(* CoDeSys 2.3.9.55 project: PLC rolety modbus.pro *)
(* Libraries: Targets\WAGO\Libraries\32_Bit\SysLibRtc.lib 8.11.10 12:37:48, Targets\WAGO\Libraries\32_Bit\Visu_Scheduler_03_e.lib 27.1.21 14:42:06, SysLibFile.lib 8.11.10 12:37:48, mod_com.lib 8.11.10 12:37:48, Targets\WAGO\Libraries\32_Bit\Scheduler_03.lib 27.1.21 14:42:05, Targets\WAGO\Libraries\32_Bit\oscat_building_100.lib 24.3.25 16:40:53, Building_common.lib 28.9.15 13:45:22, Targets\WAGO\Libraries\32_Bit\oscat_basic_333.lib 24.3.25 16:48:54, Standard.lib 8.11.10 12:37:48, SYSLIBCALLBACK.LIB 8.11.10 12:37:48 *)

(* PLC configuration (modules and I/O channels)
IN1 AT %IX0.0 [BOOLOnX_I] Biuro
IN2 AT %IX0.1 [BOOLOnX_I] Garaz
IN3 AT %IX0.2 [BOOLOnX_I] Jadalnia
IN4 AT %IX0.3 [BOOLOnX_I] Kuchnia duze
IN5 AT %IX0.4 [BOOLOnX_I] Kuchnia male
IN6 AT %IX0.5 [BOOLOnX_I] Lazienka duza
IN7 AT %IX0.6 [BOOLOnX_I] Salon duze 1
IN8 AT %IX0.7 [BOOLOnX_I] Salon duze 2
IN9 AT %IX0.8 [BOOLOnX_I] Salon taras
IN10 AT %IX0.9 [BOOLOnX_I] Schody
IN11 AT %IX0.10 [BOOLOnX_I] Sypialnia
IN12 AT %IX0.11 [BOOLOnX_I] Taras drzwi
IN13 AT %IX0.12 [BOOLOnX_I] Warsztat
IN14 AT %IX0.13 [BOOLOnX_I] rezerwa
IN15 AT %IX0.14 [BOOLOnX_I] Otworz wszystkie
IN16 AT %IX0.15 [BOOLOnX_I] Zamknij wszystkie
0750-0513 2 DO 250V AC 2.0A Rel 2NO (PotFree) [Type_10_2_Channels] node 2, in %IB1 out %QB0 {INTTypePAAssignment = PLC; INTTypeModule = plugged}
  OUTO1 AT %QX0.0 [BOOLOnX_Q] Biuro otwórz
  OUTC1 AT %QX0.1 [BOOLOnX_Q] Biuro zamknij
0750-0513 2 DO 250V AC 2.0A Rel 2NO (PotFree) [Type_10_2_Channels] node 3, in %IB2 out %QB0 {INTTypePAAssignment = PLC; INTTypeModule = plugged}
  OUTO2 AT %QX0.2 [BOOLOnX_Q] Garaz otwórz
  OUTC2 AT %QX0.3 [BOOLOnX_Q] Garaz zamknij
0750-0513 2 DO 250V AC 2.0A Rel 2NO (PotFree) [Type_10_2_Channels] node 4, in %IB2 out %QX0.2 {INTTypePAAssignment = PLC; INTTypeModule = plugged}
  OUTO3 AT %QX0.4 [BOOLOnX_Q] Jadalnia otwórz
  OUTC3 AT %QX0.5 [BOOLOnX_Q] Jadalnia zamknij
0750-0513 2 DO 250V AC 2.0A Rel 2NO (PotFree) [Type_10_2_Channels] node 5, in %IB2 out %QX0.4 {INTTypePAAssignment = PLC; INTTypeModule = plugged}
  OUTO4 AT %QX0.6 [BOOLOnX_Q] Kuchnia duze otwórz
  OUTC4 AT %QX0.7 [BOOLOnX_Q] Kuchnia duze zamknij
0750-0513 2 DO 250V AC 2.0A Rel 2NO (PotFree) [Type_10_2_Channels] node 6, in %IB2 out %QX0.6 {INTTypePAAssignment = PLC; INTTypeModule = plugged}
  OUTO5 AT %QX0.8 [BOOLOnX_Q] Kuchnia male otwórz
  OUTC5 AT %QX0.9 [BOOLOnX_Q] Kuchnia male zamknij
0750-0513 2 DO 250V AC 2.0A Rel 2NO (PotFree) [Type_10_2_Channels] node 7, in %IB2 out %QB1 {INTTypePAAssignment = PLC; INTTypeModule = plugged}
  OUTO6 AT %QX0.10 [BOOLOnX_Q] Lazienka duza otwórz
  OUTC6 AT %QX0.11 [BOOLOnX_Q] Lazienka duza zamknij
0750-0513 2 DO 250V AC 2.0A Rel 2NO (PotFree) [Type_10_2_Channels] node 8, in %IB2 out %QX0.10 {INTTypePAAssignment = PLC; INTTypeModule = plugged}
  OUTO7 AT %QX0.12 [BOOLOnX_Q] Salon duze 1 otwórz
  OUTC7 AT %QX0.13 [BOOLOnX_Q] Salon duze 1 zamknij
0750-0513 2 DO 250V AC 2.0A Rel 2NO (PotFree) [Type_10_2_Channels] node 9, in %IB2 out %QX0.12 {INTTypePAAssignment = PLC; INTTypeModule = plugged}
  OUTO8 AT %QX0.14 [BOOLOnX_Q] Salon duze 2 otwórz
  OUTC8 AT %QX0.15 [BOOLOnX_Q] Salon duze 2 zamknij
0750-0513 2 DO 250V AC 2.0A Rel 2NO (PotFree) [Type_10_2_Channels] node 10, in %IB2 out %QX0.14 {INTTypePAAssignment = PLC; INTTypeModule = plugged}
  OUTO9 AT %QX1.0 [BOOLOnX_Q] Salon taras otwórz
  OUTC9 AT %QX1.1 [BOOLOnX_Q] Salon taras zamknij
0750-0513 2 DO 250V AC 2.0A Rel 2NO (PotFree) [Type_10_2_Channels] node 11, in %IB2 out %QB2 {INTTypePAAssignment = PLC; INTTypeModule = plugged}
  OUTO10 AT %QX1.2 [BOOLOnX_Q] Schody otwórz
  OUTC10 AT %QX1.3 [BOOLOnX_Q] Schody zamknij
0750-0513 2 DO 250V AC 2.0A Rel 2NO (PotFree) [Type_10_2_Channels] node 12, in %IB2 out %QX1.2 {INTTypePAAssignment = PLC; INTTypeModule = plugged}
  OUTO11 AT %QX1.4 [BOOLOnX_Q] Sypialnia otwórz
  OUTC11 AT %QX1.5 [BOOLOnX_Q] Sypialnia zamknij
0750-0513 2 DO 250V AC 2.0A Rel 2NO (PotFree) [Type_10_2_Channels] node 13, in %IB2 out %QX1.4 {INTTypePAAssignment = PLC; INTTypeModule = plugged}
  OUTO12 AT %QX1.6 [BOOLOnX_Q] Taras otwórz
  OUTC12 AT %QX1.7 [BOOLOnX_Q] Taras zamknij
0750-0513 2 DO 250V AC 2.0A Rel 2NO (PotFree) [Type_10_2_Channels] node 14, in %IB2 out %QX1.6 {INTTypePAAssignment = PLC; INTTypeModule = plugged}
  OUTO13 AT %QX1.8 [BOOLOnX_Q] Warsztat otwórz
  OUTC13 AT %QX1.9 [BOOLOnX_Q] Warsztat zamknij
Fieldbus variables [FB_VARS] node 1, in %IB0 out %QB0
Flag variables [FLAG_VARS] node 2, in %IB0 out %QB0
Modbus-Master [MB_MASTER] node 3, in %IB0 out %QB0
*)

(* Task configuration *)
TASK Main (PRIORITY := 1); (* freewheeling *)
	PLC_PRG();
END_TASK
TASK ReadClock (PRIORITY := 10, INTERVAL := T#1000ms);
	ReadClock();
END_TASK

(* Global variable list: Global_Variables *)
VAR_GLOBAL
  CURRENT_TIME : DATE_AND_TIME;
END_VAR

(* POU PLC_PRG, ST *)
PROGRAM PLC_PRG
VAR
	(*programator tygodniowy *)
	Enable_Schedulers : BOOL := TRUE;
	Scheduler_Blind_1, Scheduler_Blind_2 : FbScheduleWeekly;
  	Scheduler_Blind_1_ON, Scheduler_Blind_2_ON : R_TRIG;
  	Scheduler_Blind_1_OFF, Scheduler_Blind_2_OFF : F_TRIG;
 	Blinds_UP, Blinds_DN : BOOL;
	(* Przyciski long/short do sterowania roletami  - 1 sec. *)
	LongShort_IN1, LongShort_IN2, LongShort_IN3, LongShort_IN4, LongShort_IN5, LongShort_IN6, LongShort_IN7, LongShort_IN8, LongShort_IN9,  LongShort_IN10,  LongShort_IN11,  LongShort_IN12,  LongShort_IN13, LongShort_IN15, LongShort_IN16 : Fb_ShortLong := (uiT_10tel_s := 10, uiTL_10tel_s := 1, uiTS_10tel_s := 1);
	(*Przyciski podwojny klik*)
	Double_IN1, Double_IN2, Double_IN3, Double_IN4, Double_IN5, Double_IN6, Double_IN7, Double_IN8, Double_IN9,  Double_IN10,  Double_IN11,  Double_IN12,  Double_IN13 : Fb_Click;
	(* Wizualizacje - Rolety *)
	VIS_Blind_1_UP,  VIS_Blind_1_DN, VIS_1_wlacz, VIS_Blind_1_SHADE : BOOL;
	VIS_Blind_2_UP,  VIS_Blind_2_DN, VIS_2_wlacz, VIS_Blind_2_SHADE : BOOL;
	VIS_Blind_3_UP,  VIS_Blind_3_DN, VIS_3_wlacz, VIS_Blind_3_SHADE : BOOL;
	VIS_Blind_4_UP,  VIS_Blind_4_DN, VIS_4_wlacz, VIS_Blind_4_SHADE : BOOL;
	VIS_Blind_5_UP,  VIS_Blind_5_DN, VIS_5_wlacz, VIS_Blind_5_SHADE : BOOL;
	VIS_Blind_6_UP,  VIS_Blind_6_DN, VIS_6_wlacz, VIS_Blind_6_SHADE : BOOL;
	VIS_Blind_7_UP,  VIS_Blind_7_DN, VIS_7_wlacz, VIS_Blind_7_SHADE : BOOL;
	VIS_Blind_8_UP,  VIS_Blind_8_DN, VIS_8_wlacz, VIS_Blind_8_SHADE : BOOL;
	VIS_Blind_9_UP,  VIS_Blind_9_DN, VIS_9_wlacz, VIS_Blind_9_SHADE : BOOL;
	VIS_Blind_10_UP,  VIS_Blind_10_DN, VIS_10_wlacz, VIS_Blind_10_SHADE : BOOL;
	VIS_Blind_11_UP,  VIS_Blind_11_DN, VIS_11_wlacz, VIS_Blind_11_SHADE : BOOL;
	VIS_Blind_12_UP,  VIS_Blind_12_DN, VIS_12_wlacz, VIS_Blind_12_SHADE : BOOL;
	VIS_Blind_13_UP,  VIS_Blind_13_DN, VIS_13_wlacz, VIS_Blind_13_SHADE : BOOL;
	(* przyciski otwórz/zamknij wszystkie *)
 	VIS_ALL_UP,  VIS_ALL_DN  : BOOL; (* do sterowania z wizualizacji *)
	(*deklaracje modbus*)
	VIS_OUT1 AT %MX294.0: BOOL;
	VIS_OUT2 AT %MX295.0: BOOL;
	VIS_OUT3 AT %MX296.0: BOOL;
	VIS_OUT4 AT %MX297.0: BOOL;
	VIS_OUT5 AT %MX298.0: BOOL;
	VIS_OUT6 AT %MX299.0: BOOL;
	VIS_OUT7 AT %MX300.0: BOOL;
	VIS_OUT8 AT %MX301.0: BOOL;
	VIS_OUT9 AT %MX302.0: BOOL;
	VIS_OUT10 AT %MX303.0: BOOL;
	VIS_OUT11 AT %MX304.0: BOOL;
	VIS_OUT12 AT %MX305.0: BOOL;
	VIS_OUT13 AT %MX306.0: BOOL;
	VIS_OUT14 AT %MX307.0: BOOL;
	VIS_OUT15 AT %MX308.0: BOOL;
	VIS_OUT16 AT %MX309.0: BOOL;
	VIS_OUT17 AT %MX310.0: BOOL;
	VIS_OUT18 AT %MX311.0: BOOL;
	VIS_OUT19 AT %MX312.0: BOOL;
	VIS_OUT20 AT %MX313.0: BOOL;
	VIS_OUT21 AT %MX314.0: BOOL;
	VIS_OUT22 AT %MX315.0: BOOL;
	VIS_OUT23 AT %MX316.0: BOOL;
	VIS_OUT24 AT %MX317.0: BOOL;
	VIS_OUT25 AT %MX318.0: BOOL;
	VIS_OUT26 AT %MX319.0: BOOL;
	VIS_OUT_ALL_UP AT %MX326.0: BOOL;
	VIS_OUT_ALL_DN AT %MX327.0: BOOL;
END_VAR
VAR RETAIN PERSISTENT
	(* Programator tygodniowy *)
	Data_Blind_1, Data_Blind_2 : typScheduleWeekly;
	(* Rolety *)
	Input_Blind_1: BLIND_INPUT := (PI := 150, MAX_RUNTIME := T#20s, MANUAL_TIMEOUT := t#60m, MASTER_MODE := TRUE);
	Control_Blind_1 : BLIND_CONTROL_S := (T_UP := T#17s, T_DN := T#17s);
	Input_Blind_2: BLIND_INPUT := (PI := 150, MAX_RUNTIME := T#35s, MANUAL_TIMEOUT := t#60m, MASTER_MODE := TRUE);
	Control_Blind_2 : BLIND_CONTROL_S := (T_UP := T#30s, T_DN := T#30s);
	Input_Blind_3: BLIND_INPUT := (PI := 150, MAX_RUNTIME := T#35s, MANUAL_TIMEOUT := t#60m, MASTER_MODE := TRUE);
	Control_Blind_3 : BLIND_CONTROL_S := (T_UP := T#30s, T_DN := T#30s);
	Input_Blind_4: BLIND_INPUT := (PI := 150, MAX_RUNTIME := T#20s, MANUAL_TIMEOUT := t#60m, MASTER_MODE := TRUE);
	Control_Blind_4 : BLIND_CONTROL_S := (T_UP := T#17s, T_DN := T#17s);
	Input_Blind_5: BLIND_INPUT := (PI := 150, MAX_RUNTIME := T#20s, MANUAL_TIMEOUT := t#60m, MASTER_MODE := TRUE);
	Control_Blind_5 : BLIND_CONTROL_S := (T_UP := T#17s, T_DN := T#17s);
	Input_Blind_6: BLIND_INPUT := (PI := 150, MAX_RUNTIME := T#35s, MANUAL_TIMEOUT := t#60m, MASTER_MODE := TRUE);
	Control_Blind_6 : BLIND_CONTROL_S := (T_UP := T#30s, T_DN := T#30s);
	Input_Blind_7: BLIND_INPUT := (PI := 150, MAX_RUNTIME := T#35s, MANUAL_TIMEOUT := t#60m, MASTER_MODE := TRUE);
	Control_Blind_7 : BLIND_CONTROL_S := (T_UP := T#30s, T_DN := T#30s);
	Input_Blind_8: BLIND_INPUT := (PI := 150, MAX_RUNTIME := T#35s, MANUAL_TIMEOUT := t#60m, MASTER_MODE := TRUE);
	Control_Blind_8 : BLIND_CONTROL_S := (T_UP := T#30s, T_DN := T#30s);
	Input_Blind_9: BLIND_INPUT := (PI := 150, MAX_RUNTIME := T#35s, MANUAL_TIMEOUT := t#60m, MASTER_MODE := TRUE);
	Control_Blind_9 : BLIND_CONTROL_S := (T_UP := T#30s, T_DN := T#30s);
	Input_Blind_10: BLIND_INPUT := (PI := 150, MAX_RUNTIME := T#20s, MANUAL_TIMEOUT := t#60m, MASTER_MODE := TRUE);
	Control_Blind_10 : BLIND_CONTROL_S := (T_UP := T#17s, T_DN := T#17s);
	Input_Blind_11: BLIND_INPUT := (PI := 150, MAX_RUNTIME := T#20s, MANUAL_TIMEOUT := t#60m, MASTER_MODE := TRUE);
	Control_Blind_11 : BLIND_CONTROL_S := (T_UP := T#17s, T_DN := T#17s);
	Input_Blind_12: BLIND_INPUT := (PI := 150, MAX_RUNTIME := T#35s, MANUAL_TIMEOUT := t#60m, MASTER_MODE := TRUE);
	Control_Blind_12 : BLIND_CONTROL_S := (T_UP := T#30s, T_DN := T#30s);
	Input_Blind_13: BLIND_INPUT := (PI := 150, MAX_RUNTIME := T#35s, MANUAL_TIMEOUT := t#60m, MASTER_MODE := TRUE);
	Control_Blind_13 : BLIND_CONTROL_S := (T_UP := T#30s, T_DN := T#30s);
	Input_Blind_ALL: BLIND_INPUT := (PI := 150, MAX_RUNTIME := T#35s, MANUAL_TIMEOUT := t#60m, MASTER_MODE := TRUE);
	Control_Blind_ALL : BLIND_CONTROL_S := (T_UP := T#30s, T_DN := T#30s);
END_VAR
(*bloki zarzadzajace timerami*)
Scheduler_Blind_1(xEnable := Enable_Schedulers, dtActualTime := CURRENT_TIME, typScheduleWeekly := Data_Blind_1);
Scheduler_Blind_2(xEnable := Enable_Schedulers, dtActualTime := CURRENT_TIME, typScheduleWeekly := Data_Blind_2);
(*wykrywanie wlaczenia/wylaczenia bloków timerów*)
Scheduler_Blind_1_ON(CLK := Scheduler_Blind_1.xSwitchChannel);
Scheduler_Blind_1_OFF(CLK := Scheduler_Blind_1.xSwitchChannel);
Scheduler_Blind_2_ON(CLK := Scheduler_Blind_2.xSwitchChannel);
Scheduler_Blind_2_OFF(CLK := Scheduler_Blind_2.xSwitchChannel);
(*sumowanie impulsów ON/OFF/Otworz-zamknij-wszystkie*)
Blinds_UP := Scheduler_Blind_1_ON.Q OR Scheduler_Blind_2_ON.Q OR VIS_ALL_UP;
Blinds_DN := Scheduler_Blind_1_OFF.Q OR Scheduler_Blind_2_OFF.Q OR VIS_ALL_DN;
(* ---------- przepianie rejestrow wejsciowych i wyjsciowych do podgladu --------------- *)
%MW100 := %IW0;
%MW200 := %QW0;
(* ---------- przyciski KRÓTKI / DLUGI --------------- *)
LongShort_IN1( xSwitch := IN1 );
LongShort_IN2( xSwitch := IN2 );
LongShort_IN3( xSwitch := IN3 );
LongShort_IN4( xSwitch := IN4 );
LongShort_IN5( xSwitch := IN5 );
LongShort_IN6( xSwitch := IN6 );
LongShort_IN7( xSwitch := IN7 );
LongShort_IN8( xSwitch := IN8 );
LongShort_IN9( xSwitch := IN9 );
LongShort_IN10( xSwitch := IN10 );
LongShort_IN11( xSwitch := IN11 );
LongShort_IN12( xSwitch := IN12 );
LongShort_IN13( xSwitch := IN13 );
LongShort_IN15( xSwitch := IN15 );
LongShort_IN16( xSwitch := IN16 );
(*Przyciski double*)
Double_IN1( xSwitch := IN1 );
Double_IN2( xSwitch := IN2 );
Double_IN3( xSwitch := IN3 );
Double_IN4( xSwitch := IN4 );
Double_IN5( xSwitch := IN5 );
Double_IN6( xSwitch := IN6 );
Double_IN7( xSwitch := IN7 );
Double_IN8( xSwitch := IN8 );
Double_IN9( xSwitch := IN9 );
Double_IN10( xSwitch := IN10 );
Double_IN11( xSwitch := IN11 );
Double_IN12( xSwitch := IN12 );
Double_IN13( xSwitch := IN13 );
(* ------------- ROLETY ------------------*)
(*Roleta Biuro*)
Input_Blind_1(
S1 := LongShort_IN1.xShort OR LongShort_IN15.xLong OR VIS_Blind_1_UP OR Blinds_UP AND VIS_1_wlacz OR VIS_OUT_ALL_UP AND VIS_1_wlacz OR VIS_OUT1,
S2 := LongShort_IN1.xLong OR LongShort_IN16.xLong OR VIS_Blind_1_DN OR Blinds_DN AND VIS_1_wlacz OR VIS_OUT_ALL_DN AND VIS_1_wlacz OR VIS_OUT2,
IN := VIS_Blind_1_SHADE OR Double_IN1.xDouble, POS := Control_Blind_1.POS
);
Control_Blind_1(
UP := Input_Blind_1.QU,
DN := Input_Blind_1.QD,
S_IN := Input_Blind_1.STATUS,
pi := Input_Blind_1.PO
);
OUTO1 := Control_Blind_1.MU;
OUTC1 := Control_Blind_1.MD;
(*Roleta Garaz*)
Input_Blind_2(
S1 := LongShort_IN2.xShort OR LongShort_IN15.xLong OR VIS_Blind_2_UP OR Blinds_UP AND VIS_2_wlacz OR VIS_OUT_ALL_UP AND VIS_2_wlacz OR VIS_OUT3,
S2 := LongShort_IN2.xLong OR LongShort_IN16.xLong OR VIS_Blind_2_DN OR Blinds_DN AND VIS_2_wlacz OR VIS_OUT_ALL_DN AND VIS_2_wlacz OR VIS_OUT4,
IN := VIS_Blind_2_SHADE OR Double_IN2.xDouble, POS := Control_Blind_2.POS
);
Control_Blind_2(
UP := Input_Blind_2.QU,
DN := Input_Blind_2.QD,
S_IN := Input_Blind_2.STATUS,
pi := Input_Blind_2.PO
);
OUTO2 := Control_Blind_2.MU;
OUTC2 := Control_Blind_2.MD;
(*Roleta Jadalnia*)
Input_Blind_3(
S1 := LongShort_IN3.xShort OR LongShort_IN15.xLong OR VIS_Blind_3_UP OR Blinds_UP AND VIS_3_wlacz OR VIS_OUT_ALL_UP AND VIS_3_wlacz OR VIS_OUT5,
S2 := LongShort_IN3.xLong OR LongShort_IN16.xLong OR VIS_Blind_3_DN OR Blinds_DN AND VIS_3_wlacz OR VIS_OUT_ALL_DN AND VIS_3_wlacz OR VIS_OUT6,
IN := VIS_Blind_3_SHADE OR Double_IN3.xDouble, POS := Control_Blind_3.POS
);
Control_Blind_3(
UP := Input_Blind_3.QU,
DN := Input_Blind_3.QD,
S_IN := Input_Blind_3.STATUS,
pi := Input_Blind_3.PO
);
OUTO3 := Control_Blind_3.MU;
OUTC3 := Control_Blind_3.MD;
(*Roleta Kuchnia duze*)
Input_Blind_4(
S1 := LongShort_IN4.xShort OR LongShort_IN15.xLong OR VIS_Blind_4_UP OR Blinds_UP AND VIS_4_wlacz OR VIS_OUT_ALL_UP AND VIS_4_wlacz OR VIS_OUT7,
S2 := LongShort_IN4.xLong OR LongShort_IN16.xLong OR VIS_Blind_4_DN OR Blinds_DN AND VIS_4_wlacz OR VIS_OUT_ALL_DN AND VIS_4_wlacz OR VIS_OUT8,
IN := VIS_Blind_4_SHADE OR Double_IN4.xDouble, POS := Control_Blind_4.POS
);
Control_Blind_4(
UP := Input_Blind_4.QU,
DN := Input_Blind_4.QD,
S_IN := Input_Blind_4.STATUS,
pi := Input_Blind_4.PO
);
OUTO4 := Control_Blind_4.MU;
OUTC4 := Control_Blind_4.MD;
(*Roleta Kuchnia male*)
Input_Blind_5(
S1 := LongShort_IN5.xShort OR LongShort_IN15.xLong OR VIS_Blind_5_UP OR Blinds_UP AND VIS_5_wlacz OR VIS_OUT_ALL_UP AND VIS_5_wlacz OR VIS_OUT9,
S2 := LongShort_IN5.xLong OR LongShort_IN16.xLong OR VIS_Blind_5_DN OR Blinds_DN AND VIS_5_wlacz OR VIS_OUT_ALL_DN AND VIS_5_wlacz OR VIS_OUT10,
IN := VIS_Blind_5_SHADE OR Double_IN5.xDouble, POS := Control_Blind_5.POS
);
Control_Blind_5(
UP := Input_Blind_5.QU,
DN := Input_Blind_5.QD,
S_IN := Input_Blind_5.STATUS,
pi := Input_Blind_5.PO
);
OUTO5 := Control_Blind_5.MU;
OUTC5 := Control_Blind_5.MD;
(*Roleta Lazienka duza*)
Input_Blind_6(
S1 := LongShort_IN6.xShort OR LongShort_IN15.xLong OR VIS_Blind_6_UP OR Blinds_UP AND VIS_6_wlacz OR VIS_OUT_ALL_UP AND VIS_6_wlacz OR VIS_OUT11,
S2 := LongShort_IN6.xLong OR LongShort_IN16.xLong OR VIS_Blind_6_DN OR Blinds_DN AND VIS_6_wlacz OR VIS_OUT_ALL_DN AND VIS_6_wlacz OR VIS_OUT12,
IN := VIS_Blind_6_SHADE OR Double_IN6.xDouble, POS := Control_Blind_6.POS
);
Control_Blind_6(
UP := Input_Blind_6.QU,
DN := Input_Blind_6.QD,
S_IN := Input_Blind_6.STATUS,
pi := Input_Blind_6.PO
);
OUTO6 := Control_Blind_6.MU;
OUTC6 := Control_Blind_6.MD;
(*Roleta Salon duze 1*)
Input_Blind_7(
S1 := LongShort_IN7.xShort OR LongShort_IN15.xLong OR VIS_Blind_7_UP OR Blinds_UP AND VIS_7_wlacz OR VIS_OUT_ALL_UP AND VIS_7_wlacz OR VIS_OUT13,
S2 := LongShort_IN7.xLong OR LongShort_IN16.xLong OR VIS_Blind_7_DN OR Blinds_DN AND VIS_7_wlacz OR VIS_OUT_ALL_DN AND VIS_7_wlacz OR VIS_OUT14,
IN := VIS_Blind_7_SHADE OR Double_IN7.xDouble, POS := Control_Blind_7.POS
);
Control_Blind_7(
UP := Input_Blind_7.QU,
DN := Input_Blind_7.QD,
S_IN := Input_Blind_7.STATUS,
pi := Input_Blind_7.PO
);
OUTO7 := Control_Blind_7.MU;
OUTC7 := Control_Blind_7.MD;
(*Roleta Salon duze 2*)
Input_Blind_8(
S1 := LongShort_IN8.xShort OR LongShort_IN15.xLong OR VIS_Blind_8_UP OR Blinds_UP AND VIS_8_wlacz OR VIS_OUT_ALL_UP AND VIS_8_wlacz OR VIS_OUT15,
S2 := LongShort_IN8.xLong OR LongShort_IN16.xLong OR VIS_Blind_8_DN OR Blinds_DN AND VIS_8_wlacz OR VIS_OUT_ALL_DN AND VIS_8_wlacz OR VIS_OUT16,
IN := VIS_Blind_8_SHADE OR Double_IN8.xDouble, POS := Control_Blind_8.POS
);
Control_Blind_8(
UP := Input_Blind_8.QU,
DN := Input_Blind_8.QD,
S_IN := Input_Blind_8.STATUS,
pi := Input_Blind_8.PO
);
OUTO8 := Control_Blind_8.MU;
OUTC8 := Control_Blind_8.MD;
(*Roleta  Salon taras*)
Input_Blind_9(
S1 := LongShort_IN9.xShort OR LongShort_IN15.xLong OR VIS_Blind_9_UP OR Blinds_UP AND VIS_9_wlacz OR VIS_OUT_ALL_UP AND VIS_9_wlacz OR VIS_OUT17,
S2 := LongShort_IN9.xLong OR LongShort_IN16.xLong OR VIS_Blind_9_DN OR Blinds_DN AND VIS_9_wlacz OR VIS_OUT_ALL_DN AND VIS_9_wlacz OR VIS_OUT18,
IN := VIS_Blind_9_SHADE OR Double_IN9.xDouble, POS := Control_Blind_9.POS
);
Control_Blind_9(
UP := Input_Blind_9.QU,
DN := Input_Blind_9.QD,
S_IN := Input_Blind_9.STATUS,
pi := Input_Blind_9.PO
);
OUTO9 := Control_Blind_9.MU;
OUTC9 := Control_Blind_9.MD;
(*Roleta schody*)
Input_Blind_10(
S1 := LongShort_IN10.xShort OR LongShort_IN15.xLong OR VIS_Blind_10_UP OR Blinds_UP AND VIS_10_wlacz OR VIS_OUT_ALL_UP AND VIS_10_wlacz OR VIS_OUT19,
S2 := LongShort_IN10.xLong OR LongShort_IN16.xLong OR VIS_Blind_10_DN OR Blinds_DN AND VIS_10_wlacz OR VIS_OUT_ALL_DN AND VIS_10_wlacz OR VIS_OUT20,
IN := VIS_Blind_10_SHADE OR Double_IN10.xDouble, POS := Control_Blind_10.POS
);
Control_Blind_10(
UP := Input_Blind_10.QU,
DN := Input_Blind_10.QD,
S_IN := Input_Blind_10.STATUS,
pi := Input_Blind_10.PO
);
OUTO10 := Control_Blind_10.MU;
OUTC10 := Control_Blind_10.MD;
(*Roleta sypialnia*)
Input_Blind_11(
S1 := LongShort_IN11.xShort OR LongShort_IN15.xLong OR VIS_Blind_11_UP OR Blinds_UP AND VIS_11_wlacz OR VIS_OUT_ALL_UP AND VIS_11_wlacz OR VIS_OUT21,
S2 := LongShort_IN11.xLong OR LongShort_IN16.xLong OR VIS_Blind_11_DN OR Blinds_DN AND VIS_11_wlacz OR VIS_OUT_ALL_DN AND VIS_11_wlacz OR VIS_OUT22,
IN := VIS_Blind_11_SHADE OR Double_IN11.xDouble, POS := Control_Blind_11.POS
);
Control_Blind_11(
UP := Input_Blind_11.QU,
DN := Input_Blind_11.QD,
S_IN := Input_Blind_11.STATUS,
pi := Input_Blind_11.PO
);
OUTO11 := Control_Blind_11.MU;
OUTC11 := Control_Blind_11.MD;
(*Roleta taras drzwi*)
Input_Blind_12(
S1 := LongShort_IN12.xShort OR LongShort_IN15.xLong OR VIS_Blind_12_UP OR Blinds_UP AND VIS_12_wlacz OR VIS_OUT_ALL_UP AND VIS_12_wlacz OR VIS_OUT23,
S2 := LongShort_IN12.xLong OR LongShort_IN16.xLong OR VIS_Blind_12_DN OR Blinds_DN AND VIS_12_wlacz OR VIS_OUT_ALL_DN AND VIS_12_wlacz OR VIS_OUT24,
IN := VIS_Blind_12_SHADE OR Double_IN12.xDouble, POS := Control_Blind_12.POS
);
Control_Blind_12(
UP := Input_Blind_12.QU,
DN := Input_Blind_12.QD,
S_IN := Input_Blind_12.STATUS,
pi := Input_Blind_12.PO
);
OUTO12 := Control_Blind_12.MU;
OUTC12 := Control_Blind_12.MD;
(*Roleta warsztat*)
Input_Blind_13(
S1 := LongShort_IN13.xShort OR LongShort_IN15.xLong OR VIS_Blind_13_UP OR Blinds_UP AND VIS_13_wlacz OR VIS_OUT_ALL_UP AND VIS_13_wlacz OR VIS_OUT25,
S2 := LongShort_IN13.xLong OR LongShort_IN16.xLong OR VIS_Blind_13_DN OR Blinds_DN AND VIS_13_wlacz OR VIS_OUT_ALL_DN AND VIS_13_wlacz OR VIS_OUT26,
IN := VIS_Blind_13_SHADE OR Double_IN13.xDouble, POS := Control_Blind_13.POS
);
Control_Blind_13(
UP := Input_Blind_13.QU,
DN := Input_Blind_13.QD,
S_IN := Input_Blind_13.STATUS,
pi := Input_Blind_13.PO
);
OUTO13 := Control_Blind_13.MU;
OUTC13 := Control_Blind_13.MD;
(*modbus zerowanie zmiennej*)
IF VIS_OUT_ALL_DN THEN
VIS_OUT_ALL_DN := 0;
END_IF
IF VIS_OUT_ALL_UP THEN
VIS_OUT_ALL_UP := 0;
END_IF
IF VIS_OUT1 THEN
VIS_OUT1 := 0;
END_IF
IF VIS_OUT2 THEN
VIS_OUT2 := 0;
END_IF
IF VIS_OUT3 THEN
VIS_OUT3 := 0;
END_IF
IF VIS_OUT4 THEN
VIS_OUT4 := 0;
END_IF
IF VIS_OUT5 THEN
VIS_OUT5 := 0;
END_IF
IF VIS_OUT6 THEN
VIS_OUT6 := 0;
END_IF
IF VIS_OUT7 THEN
VIS_OUT7 := 0;
END_IF
IF VIS_OUT8 THEN
VIS_OUT8 := 0;
END_IF
IF VIS_OUT9 THEN
VIS_OUT9 := 0;
END_IF
IF VIS_OUT10 THEN
VIS_OUT10 := 0;
END_IF
IF VIS_OUT11 THEN
VIS_OUT11 := 0;
END_IF
IF VIS_OUT12 THEN
VIS_OUT12 := 0;
END_IF
IF VIS_OUT13 THEN
VIS_OUT13 := 0;
END_IF
IF VIS_OUT14 THEN
VIS_OUT14 := 0;
END_IF
IF VIS_OUT15 THEN
VIS_OUT15 := 0;
END_IF
IF VIS_OUT16 THEN
VIS_OUT16 := 0;
END_IF
IF VIS_OUT17 THEN
VIS_OUT17 := 0;
END_IF
IF VIS_OUT18 THEN
VIS_OUT18 := 0;
END_IF
IF VIS_OUT19 THEN
VIS_OUT19 := 0;
END_IF
IF VIS_OUT20 THEN
VIS_OUT20 := 0;
END_IF
IF VIS_OUT21 THEN
VIS_OUT21 := 0;
END_IF
IF VIS_OUT22 THEN
VIS_OUT22 := 0;
END_IF
IF VIS_OUT23 THEN
VIS_OUT23 := 0;
END_IF
IF VIS_OUT24 THEN
VIS_OUT24 := 0;
END_IF
IF VIS_OUT25 THEN
VIS_OUT25 := 0;
END_IF
IF VIS_OUT26 THEN
VIS_OUT26 := 0;
END_IF
END_PROGRAM

(* POU ReadClock, ST *)
PROGRAM ReadClock
VAR
END_VAR
CURRENT_TIME := SysRtcGetTime(TRUE);
END_PROGRAM

(* POU Configuration/MODBUS_CONFIGURATION, ST *)
PROGRAM MODBUS_CONFIGURATION
VAR                                
END_VAR                            
(*
   <?xml version="1.0" encoding="UTF-16" standalone="yes"?>
<network xml_structure_version="1" xml_feature_version="1">
	<generator_settings minRTUTaskCycleTimeMs="5" minEthaskCycleTimeMs="5" ethSlaveMultiplier="0.1" rtuInterfaceMultiplier="0.1" taskGeneration="true"/>
</network>
                              
*)                                 
;
END_PROGRAM

(* Visualisation harmonogram
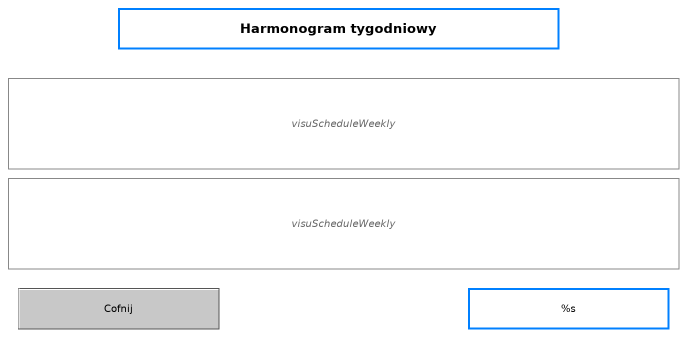
rounded rectangle at (470,300)-(671,341): text "%s"; shows CURRENT_TIME
embedded screen at (10,90)-(681,181): visuScheduleWeekly
embedded screen at (10,190)-(681,281): visuScheduleWeekly
rounded rectangle at (120,20)-(561,61): text "Harmonogram tygodniowy"
button at (20,300)-(221,341): text "Cofnij"; opens PLC_VISU
*)

(* Visualisation PLC_VISU
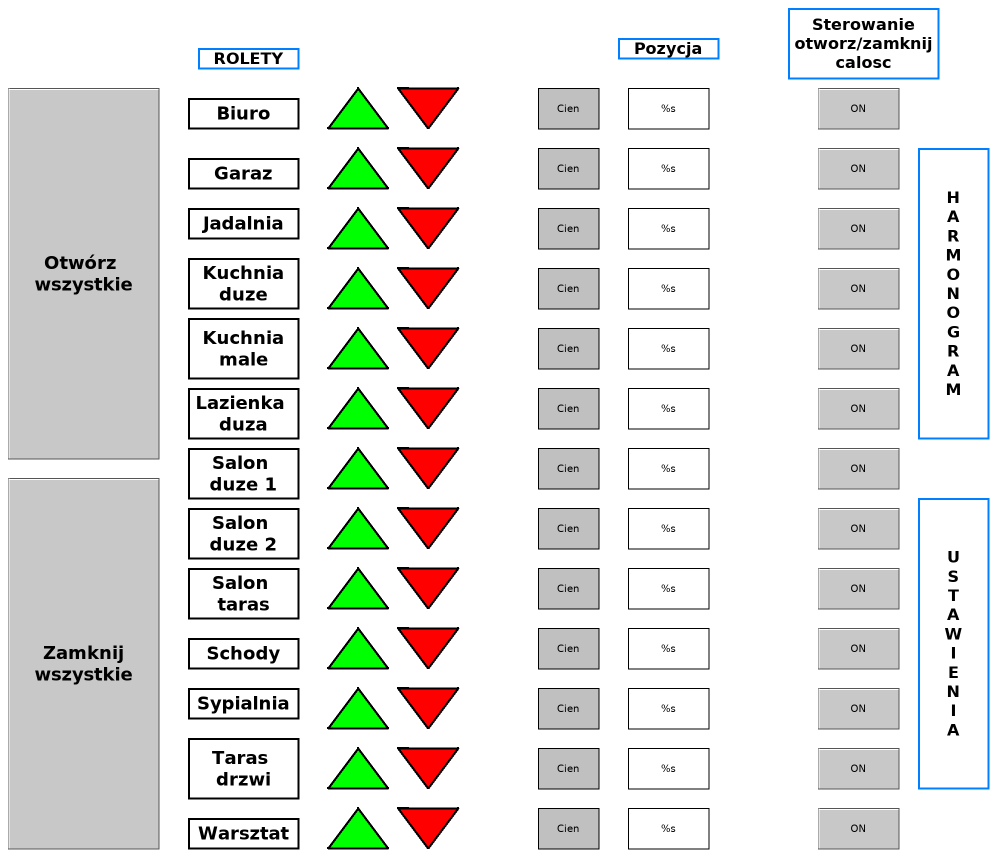
rounded rectangle at (540,440)-(601,481): text "Cien"; taps PLC_PRG.VIS_Blind_7_SHADE
rounded rectangle at (540,500)-(601,541): text "Cien"; taps PLC_PRG.VIS_Blind_8_SHADE
rounded rectangle at (630,440)-(711,481): text "%s"; shows PLC_PRG.Control_Blind_7.POS
rounded rectangle at (630,500)-(711,541): text "%s"; shows PLC_PRG.Control_Blind_8.POS
rounded rectangle at (190,440)-(301,491): text "Salon / duze 1"
rounded rectangle at (190,500)-(301,551): text "Salon / duze 2"
rounded rectangle at (540,380)-(601,421): text "Cien"; taps PLC_PRG.VIS_Blind_6_SHADE
rounded rectangle at (630,380)-(711,421): text "%s"; shows PLC_PRG.Control_Blind_6.POS
rounded rectangle at (540,320)-(601,361): text "Cien"; taps PLC_PRG.VIS_Blind_5_SHADE
rounded rectangle at (630,320)-(711,361): text "%s"; shows PLC_PRG.Control_Blind_5.POS
rounded rectangle at (540,260)-(601,301): text "Cien"; taps PLC_PRG.VIS_Blind_4_SHADE
rounded rectangle at (630,260)-(711,301): text "%s"; shows PLC_PRG.Control_Blind_4.POS
rounded rectangle at (540,200)-(601,241): text "Cien"; taps PLC_PRG.VIS_Blind_3_SHADE
rounded rectangle at (630,200)-(711,241): text "%s"; shows PLC_PRG.Control_Blind_3.POS
rounded rectangle at (540,140)-(601,181): text "Cien"; taps PLC_PRG.VIS_Blind_2_SHADE
rounded rectangle at (630,140)-(711,181): text "%s"; shows PLC_PRG.Control_Blind_2.POS
rounded rectangle at (540,560)-(601,601): text "Cien"; taps PLC_PRG.VIS_Blind_9_SHADE
rounded rectangle at (630,560)-(711,601): text "%s"; shows PLC_PRG.Control_Blind_9.POS
rounded rectangle at (540,80)-(601,121): text "Cien"; taps PLC_PRG.VIS_Blind_1_SHADE
rounded rectangle at (630,80)-(711,121): text "%s"; shows PLC_PRG.Control_Blind_1.POS
rounded rectangle at (190,560)-(301,611): text "Salon / taras"
rounded rectangle at (190,380)-(301,431): text "Lazienka / duza"
rounded rectangle at (190,310)-(301,371): text "Kuchnia / male"
rounded rectangle at (190,250)-(301,301): text "Kuchnia / duze"
rounded rectangle at (190,200)-(301,231): text "Jadalnia"
rounded rectangle at (190,150)-(301,181): text "Garaz"
rounded rectangle at (190,90)-(301,121): text "Biuro"
rounded rectangle at (200,40)-(301,61): text "ROLETY"
rounded rectangle at (620,30)-(721,51): text "Pozycja"
rounded rectangle at (540,620)-(601,661): text "Cien"; taps PLC_PRG.VIS_Blind_10_SHADE
rounded rectangle at (630,620)-(711,661): text "%s"; shows PLC_PRG.Control_Blind_10.POS
rounded rectangle at (190,630)-(301,661): text "Schody"
rounded rectangle at (540,680)-(601,721): text "Cien"; taps PLC_PRG.VIS_Blind_11_SHADE
rounded rectangle at (630,680)-(711,721): text "%s"; shows PLC_PRG.Control_Blind_11.POS
rounded rectangle at (190,680)-(301,711): text "Sypialnia"
rounded rectangle at (540,740)-(601,781): text "Cien"; taps PLC_PRG.VIS_Blind_12_SHADE
rounded rectangle at (630,740)-(711,781): text "%s"; shows PLC_PRG.Control_Blind_12.POS
rounded rectangle at (190,730)-(301,791): text "Taras / drzwi"
rounded rectangle at (540,800)-(601,841): text "Cien"; taps PLC_PRG.VIS_Blind_13_SHADE
rounded rectangle at (630,800)-(711,841): text "%s"; shows PLC_PRG.Control_Blind_13.POS
rounded rectangle at (190,810)-(301,841): text "Warsztat"
polygon at (330,80)-(390,120): alarm colour if OUTO1; taps PLC_PRG.VIS_Blind_1_UP
polygon at (400,80)-(460,120): alarm colour if OUTC1; taps PLC_PRG.VIS_Blind_1_DN
polygon at (330,140)-(390,180): alarm colour if OUTO2; taps PLC_PRG.VIS_Blind_2_UP
polygon at (400,140)-(460,180): alarm colour if OUTC2; taps PLC_PRG.VIS_Blind_2_DN
polygon at (330,200)-(390,240): alarm colour if OUTO3; taps PLC_PRG.VIS_Blind_3_UP
polygon at (400,200)-(460,240): alarm colour if OUTC3; taps PLC_PRG.VIS_Blind_3_DN
polygon at (330,260)-(390,300): alarm colour if OUTO4; taps PLC_PRG.VIS_Blind_4_UP
polygon at (400,260)-(460,300): alarm colour if OUTC4; taps PLC_PRG.VIS_Blind_4_DN
polygon at (330,320)-(390,360): alarm colour if OUTO5; taps PLC_PRG.VIS_Blind_5_UP
polygon at (400,320)-(460,360): alarm colour if OUTC5; taps PLC_PRG.VIS_Blind_5_DN
polygon at (330,380)-(390,420): alarm colour if OUTO6; taps PLC_PRG.VIS_Blind_6_UP
polygon at (400,380)-(460,420): alarm colour if OUTC6; taps PLC_PRG.VIS_Blind_6_DN
polygon at (330,440)-(390,480): alarm colour if OUTO7; taps PLC_PRG.VIS_Blind_7_UP
polygon at (400,440)-(460,480): alarm colour if OUTC7; taps PLC_PRG.VIS_Blind_7_DN
polygon at (330,500)-(390,540): alarm colour if OUTO8; taps PLC_PRG.VIS_Blind_8_UP
polygon at (400,500)-(460,540): alarm colour if OUTC8; taps PLC_PRG.VIS_Blind_8_DN
polygon at (330,560)-(390,600): alarm colour if OUTO9; taps PLC_PRG.VIS_Blind_9_UP
polygon at (400,560)-(460,600): alarm colour if OUTC9; taps PLC_PRG.VIS_Blind_9_DN
polygon at (330,620)-(390,660): alarm colour if OUTO10; taps PLC_PRG.VIS_Blind_10_UP
polygon at (400,620)-(460,660): alarm colour if OUTC10; taps PLC_PRG.VIS_Blind_10_DN
polygon at (330,680)-(390,720): alarm colour if OUTO11; taps PLC_PRG.VIS_Blind_11_UP
polygon at (400,680)-(460,720): alarm colour if OUTC11; taps PLC_PRG.VIS_Blind_11_DN
polygon at (330,740)-(390,780): alarm colour if OUTO12; taps PLC_PRG.VIS_Blind_12_UP
polygon at (400,740)-(460,780): alarm colour if OUTC12; taps PLC_PRG.VIS_Blind_12_DN
polygon at (330,800)-(390,840): alarm colour if OUTO13; taps PLC_PRG.VIS_Blind_13_UP
polygon at (400,800)-(460,840): alarm colour if OUTC13; taps PLC_PRG.VIS_Blind_13_DN
button at (10,80)-(161,451): text "Otwórz / wszystkie"; taps PLC_PRG.VIS_ALL_UP
button at (10,470)-(161,841): text "Zamknij / wszystkie"; taps PLC_PRG.VIS_ALL_DN
button at (820,80)-(901,121): text "ON"; toggles PLC_PRG.VIS_1_wlacz
button at (820,140)-(901,181): text "ON"; toggles PLC_PRG.VIS_2_wlacz
button at (820,200)-(901,241): text "ON"; toggles PLC_PRG.VIS_3_wlacz
button at (820,260)-(901,301): text "ON"; toggles PLC_PRG.VIS_4_wlacz
button at (820,320)-(901,361): text "ON"; toggles PLC_PRG.VIS_5_wlacz
button at (820,380)-(901,421): text "ON"; toggles PLC_PRG.VIS_6_wlacz
button at (820,440)-(901,481): text "ON"; toggles PLC_PRG.VIS_7_wlacz
button at (820,500)-(901,541): text "ON"; toggles PLC_PRG.VIS_8_wlacz
button at (820,560)-(901,601): text "ON"; toggles PLC_PRG.VIS_9_wlacz
button at (820,620)-(901,661): text "ON"; toggles PLC_PRG.VIS_10_wlacz
button at (820,680)-(901,721): text "ON"; toggles PLC_PRG.VIS_11_wlacz
button at (820,740)-(901,781): text "ON"; toggles PLC_PRG.VIS_12_wlacz
button at (820,800)-(901,841): text "ON"; toggles PLC_PRG.VIS_13_wlacz
rounded rectangle at (790,0)-(941,71): text "Sterowanie / otworz/zamknij / calosc"
rounded rectangle at (920,140)-(991,431): text "H / A / R / M / O / N / O / G / R / A / M"; opens harmonogram
rounded rectangle at (920,490)-(991,781): text "U / S / T / A / W / I / E / N / I / A"; opens ustawienia
*)

(* Visualisation ustawienia
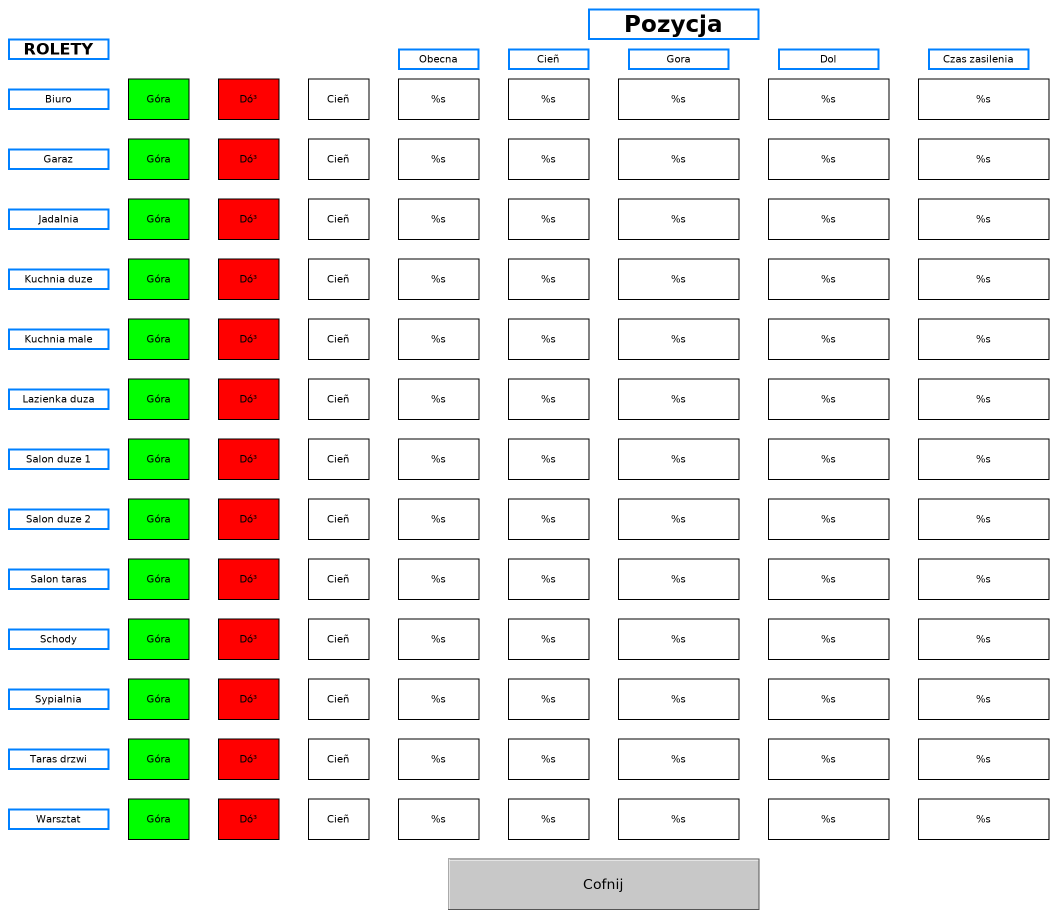
rectangle at (240,440)-(301,481): text "Góra"; alarm colour if OUTO7; taps PLC_PRG.VIS_Blind_7_UP
rectangle at (240,500)-(301,541): text "Góra"; alarm colour if OUTO8; taps PLC_PRG.VIS_Blind_8_UP
rectangle at (330,440)-(391,481): text "Dó³"; alarm colour if OUTC7; taps PLC_PRG.VIS_Blind_7_DN
rectangle at (330,500)-(391,541): text "Dó³"; alarm colour if OUTC8; taps PLC_PRG.VIS_Blind_8_DN
rectangle at (420,440)-(481,481): text "Cieñ"; taps PLC_PRG.VIS_Blind_7_SHADE
rectangle at (420,500)-(481,541): text "Cieñ"; taps PLC_PRG.VIS_Blind_8_SHADE
rectangle at (510,440)-(591,481): text "%s"; shows PLC_PRG.Control_Blind_7.POS
rectangle at (510,500)-(591,541): text "%s"; shows PLC_PRG.Control_Blind_8.POS
rectangle at (620,440)-(701,481): text "%s"; shows PLC_PRG.Input_Blind_7.PI; editable
rectangle at (620,500)-(701,541): text "%s"; shows PLC_PRG.Input_Blind_8.PI; editable
rectangle at (730,440)-(851,481): text "%s"; shows PLC_PRG.Control_Blind_7.T_UP; editable
rectangle at (730,500)-(851,541): text "%s"; shows PLC_PRG.Control_Blind_8.T_UP; editable
rectangle at (880,440)-(1001,481): text "%s"; shows PLC_PRG.Control_Blind_7.T_DN; editable
rectangle at (880,500)-(1001,541): text "%s"; shows PLC_PRG.Control_Blind_8.T_DN; editable
rectangle at (1030,440)-(1161,481): text "%s"; shows PLC_PRG.Input_Blind_7.MAX_RUNTIME; editable
rectangle at (1030,500)-(1161,541): text "%s"; shows PLC_PRG.Input_Blind_8.MAX_RUNTIME; editable
rectangle at (120,450)-(221,471): text "Salon duze 1"
rounded rectangle at (120,510)-(221,531): text "Salon duze 2"
rectangle at (240,380)-(301,421): text "Góra"; alarm colour if OUTO6; taps PLC_PRG.VIS_Blind_6_UP
rectangle at (330,380)-(391,421): text "Dó³"; alarm colour if OUTC6; taps PLC_PRG.VIS_Blind_6_DN
rectangle at (420,380)-(481,421): text "Cieñ"; taps PLC_PRG.VIS_Blind_6_SHADE
rectangle at (510,380)-(591,421): text "%s"; shows PLC_PRG.Control_Blind_6.POS
rectangle at (620,380)-(701,421): text "%s"; shows PLC_PRG.Input_Blind_6.PI; editable
rectangle at (730,380)-(851,421): text "%s"; shows PLC_PRG.Control_Blind_6.T_UP; editable
rectangle at (880,380)-(1001,421): text "%s"; shows PLC_PRG.Control_Blind_6.T_DN; editable
rectangle at (1030,380)-(1161,421): text "%s"; shows PLC_PRG.Input_Blind_6.MAX_RUNTIME; editable
rectangle at (240,320)-(301,361): text "Góra"; alarm colour if OUTO5; taps PLC_PRG.VIS_Blind_5_UP
rectangle at (330,320)-(391,361): text "Dó³"; alarm colour if OUTC5; taps PLC_PRG.VIS_Blind_5_DN
rectangle at (420,320)-(481,361): text "Cieñ"; taps PLC_PRG.VIS_Blind_5_SHADE
rectangle at (510,320)-(591,361): text "%s"; shows PLC_PRG.Control_Blind_5.POS
rectangle at (620,320)-(701,361): text "%s"; shows PLC_PRG.Input_Blind_5.PI; editable
rectangle at (730,320)-(851,361): text "%s"; shows PLC_PRG.Control_Blind_5.T_UP; editable
rectangle at (880,320)-(1001,361): text "%s"; shows PLC_PRG.Control_Blind_5.T_DN; editable
rectangle at (1030,320)-(1161,361): text "%s"; shows PLC_PRG.Input_Blind_5.MAX_RUNTIME; editable
rectangle at (240,260)-(301,301): text "Góra"; alarm colour if OUTO4; taps PLC_PRG.VIS_Blind_4_UP
rectangle at (330,260)-(391,301): text "Dó³"; alarm colour if OUTC4; taps PLC_PRG.VIS_Blind_4_DN
rectangle at (420,260)-(481,301): text "Cieñ"; taps PLC_PRG.VIS_Blind_4_SHADE
rectangle at (510,260)-(591,301): text "%s"; shows PLC_PRG.Control_Blind_4.POS
rectangle at (620,260)-(701,301): text "%s"; shows PLC_PRG.Input_Blind_4.PI; editable
rectangle at (730,260)-(851,301): text "%s"; shows PLC_PRG.Control_Blind_4.T_UP; editable
rectangle at (880,260)-(1001,301): text "%s"; shows PLC_PRG.Control_Blind_4.T_DN; editable
rectangle at (1030,260)-(1161,301): text "%s"; shows PLC_PRG.Input_Blind_4.MAX_RUNTIME; editable
rectangle at (240,200)-(301,241): text "Góra"; alarm colour if OUTO3; taps PLC_PRG.VIS_Blind_3_UP
rectangle at (330,200)-(391,241): text "Dó³"; alarm colour if OUTC3; taps PLC_PRG.VIS_Blind_3_DN
rectangle at (420,200)-(481,241): text "Cieñ"; taps PLC_PRG.VIS_Blind_3_SHADE
rectangle at (510,200)-(591,241): text "%s"; shows PLC_PRG.Control_Blind_3.POS
rectangle at (620,200)-(701,241): text "%s"; shows PLC_PRG.Input_Blind_3.PI; editable
rectangle at (730,200)-(851,241): text "%s"; shows PLC_PRG.Control_Blind_3.T_UP; editable
rectangle at (880,200)-(1001,241): text "%s"; shows PLC_PRG.Control_Blind_3.T_DN; editable
rectangle at (1030,200)-(1161,241): text "%s"; shows PLC_PRG.Input_Blind_3.MAX_RUNTIME; editable
rectangle at (240,140)-(301,181): text "Góra"; alarm colour if OUTO2; taps PLC_PRG.VIS_Blind_2_UP
rectangle at (330,140)-(391,181): text "Dó³"; alarm colour if OUTC2; taps PLC_PRG.VIS_Blind_2_DN
rectangle at (420,140)-(481,181): text "Cieñ"; taps PLC_PRG.VIS_Blind_2_SHADE
rectangle at (510,140)-(591,181): text "%s"; shows PLC_PRG.Control_Blind_2.POS
rectangle at (620,140)-(701,181): text "%s"; shows PLC_PRG.Input_Blind_2.PI; editable
rectangle at (730,140)-(851,181): text "%s"; shows PLC_PRG.Control_Blind_2.T_UP; editable
rectangle at (880,140)-(1001,181): text "%s"; shows PLC_PRG.Control_Blind_2.T_DN; editable
rectangle at (1030,140)-(1161,181): text "%s"; shows PLC_PRG.Input_Blind_2.MAX_RUNTIME; editable
rectangle at (240,560)-(301,601): text "Góra"; alarm colour if OUTO9; taps PLC_PRG.VIS_Blind_9_UP
rectangle at (330,560)-(391,601): text "Dó³"; alarm colour if OUTC9; taps PLC_PRG.VIS_Blind_9_DN
rectangle at (420,560)-(481,601): text "Cieñ"; taps PLC_PRG.VIS_Blind_9_SHADE
rectangle at (510,560)-(591,601): text "%s"; shows PLC_PRG.Control_Blind_9.POS
rectangle at (620,560)-(701,601): text "%s"; shows PLC_PRG.Input_Blind_9.PI; editable
rectangle at (730,560)-(851,601): text "%s"; shows PLC_PRG.Control_Blind_9.T_UP; editable
rectangle at (880,560)-(1001,601): text "%s"; shows PLC_PRG.Control_Blind_9.T_DN; editable
rectangle at (1030,560)-(1161,601): text "%s"; shows PLC_PRG.Input_Blind_9.MAX_RUNTIME; editable
rectangle at (240,80)-(301,121): text "Góra"; alarm colour if OUTO1; taps PLC_PRG.VIS_Blind_1_UP
rectangle at (330,80)-(391,121): text "Dó³"; alarm colour if OUTC1; taps PLC_PRG.VIS_Blind_1_DN
rectangle at (420,80)-(481,121): text "Cieñ"; taps PLC_PRG.VIS_Blind_1_SHADE
rectangle at (510,80)-(591,121): text "%s"; shows PLC_PRG.Control_Blind_1.POS
rectangle at (620,80)-(701,121): text "%s"; shows PLC_PRG.Input_Blind_1.PI; editable
rectangle at (730,80)-(851,121): text "%s"; shows PLC_PRG.Control_Blind_1.T_UP; editable
rectangle at (880,80)-(1001,121): text "%s"; shows PLC_PRG.Control_Blind_1.T_DN; editable
rectangle at (1030,80)-(1161,121): text "%s"; shows PLC_PRG.Input_Blind_1.MAX_RUNTIME; editable
rounded rectangle at (120,570)-(221,591): text "Salon taras"
rectangle at (120,390)-(221,411): text "Lazienka duza"
rounded rectangle at (120,330)-(221,351): text "Kuchnia male"
rectangle at (120,270)-(221,291): text "Kuchnia duze"
rounded rectangle at (120,210)-(221,231): text "Jadalnia"
rounded rectangle at (120,150)-(221,171): text "Garaz"
rounded rectangle at (120,90)-(221,111): text "Biuro"
rounded rectangle at (120,40)-(221,61): text "ROLETY"
rounded rectangle at (510,50)-(591,71): text "Obecna"
rounded rectangle at (620,50)-(701,71): text "Cieñ"
rounded rectangle at (700,10)-(871,41): text "Pozycja"
rounded rectangle at (740,50)-(841,71): text "Gora"
rounded rectangle at (890,50)-(991,71): text "Dol"
rectangle at (1040,50)-(1141,71): text "Czas zasilenia"
rectangle at (240,620)-(301,661): text "Góra"; alarm colour if OUTO10; taps PLC_PRG.VIS_Blind_10_UP
rectangle at (330,620)-(391,661): text "Dó³"; alarm colour if OUTC10; taps PLC_PRG.VIS_Blind_10_DN
rectangle at (420,620)-(481,661): text "Cieñ"; taps PLC_PRG.VIS_Blind_10_SHADE
rectangle at (510,620)-(591,661): text "%s"; shows PLC_PRG.Control_Blind_10.POS
rectangle at (620,620)-(701,661): text "%s"; shows PLC_PRG.Input_Blind_10.PI; editable
rectangle at (730,620)-(851,661): text "%s"; shows PLC_PRG.Control_Blind_10.T_UP; editable
rectangle at (880,620)-(1001,661): text "%s"; shows PLC_PRG.Control_Blind_10.T_DN; editable
rectangle at (1030,620)-(1161,661): text "%s"; shows PLC_PRG.Input_Blind_10.MAX_RUNTIME; editable
rounded rectangle at (120,630)-(221,651): text "Schody"
rectangle at (240,680)-(301,721): text "Góra"; alarm colour if OUTO11; taps PLC_PRG.VIS_Blind_11_UP
rectangle at (330,680)-(391,721): text "Dó³"; alarm colour if OUTC11; taps PLC_PRG.VIS_Blind_11_DN
rectangle at (420,680)-(481,721): text "Cieñ"; taps PLC_PRG.VIS_Blind_11_SHADE
rectangle at (510,680)-(591,721): text "%s"; shows PLC_PRG.Control_Blind_11.POS
rectangle at (620,680)-(701,721): text "%s"; shows PLC_PRG.Input_Blind_11.PI; editable
rectangle at (730,680)-(851,721): text "%s"; shows PLC_PRG.Control_Blind_11.T_UP; editable
rectangle at (880,680)-(1001,721): text "%s"; shows PLC_PRG.Control_Blind_11.T_DN; editable
rectangle at (1030,680)-(1161,721): text "%s"; shows PLC_PRG.Input_Blind_11.MAX_RUNTIME; editable
rounded rectangle at (120,690)-(221,711): text "Sypialnia"
rectangle at (240,740)-(301,781): text "Góra"; alarm colour if OUTO12; taps PLC_PRG.VIS_Blind_12_UP
rectangle at (330,740)-(391,781): text "Dó³"; alarm colour if OUTC12; taps PLC_PRG.VIS_Blind_12_DN
rectangle at (420,740)-(481,781): text "Cieñ"; taps PLC_PRG.VIS_Blind_12_SHADE
rectangle at (510,740)-(591,781): text "%s"; shows PLC_PRG.Control_Blind_12.POS
rectangle at (620,740)-(701,781): text "%s"; shows PLC_PRG.Input_Blind_12.PI; editable
rectangle at (730,740)-(851,781): text "%s"; shows PLC_PRG.Control_Blind_12.T_UP; editable
rectangle at (880,740)-(1001,781): text "%s"; shows PLC_PRG.Control_Blind_12.T_DN; editable
rectangle at (1030,740)-(1161,781): text "%s"; shows PLC_PRG.Input_Blind_12.MAX_RUNTIME; editable
rounded rectangle at (120,750)-(221,771): text "Taras drzwi"
rectangle at (240,800)-(301,841): text "Góra"; alarm colour if OUTO13; taps PLC_PRG.VIS_Blind_13_UP
rectangle at (330,800)-(391,841): text "Dó³"; alarm colour if OUTC13; taps PLC_PRG.VIS_Blind_13_DN
rectangle at (420,800)-(481,841): text "Cieñ"; taps PLC_PRG.VIS_Blind_13_SHADE
rectangle at (510,800)-(591,841): text "%s"; shows PLC_PRG.Control_Blind_13.POS
rectangle at (620,800)-(701,841): text "%s"; shows PLC_PRG.Input_Blind_13.PI; editable
rectangle at (730,800)-(851,841): text "%s"; shows PLC_PRG.Control_Blind_13.T_UP; editable
rectangle at (880,800)-(1001,841): text "%s"; shows PLC_PRG.Control_Blind_13.T_DN; editable
rectangle at (1030,800)-(1161,841): text "%s"; shows PLC_PRG.Input_Blind_13.MAX_RUNTIME; editable
rounded rectangle at (120,810)-(221,831): text "Warsztat"
button at (560,860)-(871,911): text "Cofnij"; opens PLC_VISU
*)
